// Mitsubishi GX Developer project: 11-702日式面打機_201109261430   PLC: FX1S

PROGRAM MAIN
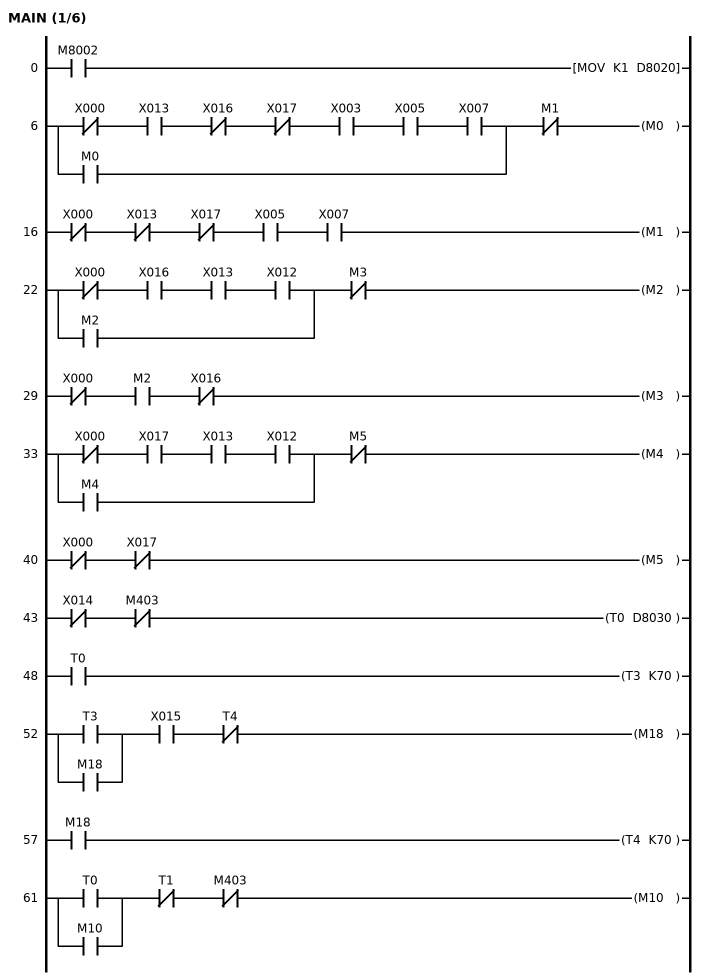
0     LD      M8002
      MOV     K1 D8020
6     LDI     X000
      AND     X013
      ANI     X016
      ANI     X017
      AND     X003
      AND     X005
      AND     X007
      OR      M0
      ANI     M1
      OUT     M0
16    LDI     X000
      ANI     X013
      ANI     X017
      AND     X005
      AND     X007
      OUT     M1
22    LDI     X000
      AND     X016
      AND     X013
      AND     X012
      OR      M2
      ANI     M3
      OUT     M2
29    LDI     X000
      AND     M2
      ANI     X016
      OUT     M3
33    LDI     X000
      AND     X017
      AND     X013
      AND     X012
      OR      M4
      ANI     M5
      OUT     M4
40    LDI     X000
      ANI     X017
      OUT     M5
43    LDI     X014
      ANI     M403
      OUT     T0 D8030
48    LD      T0
      OUT     T3 K70
52    LD      T3
      OR      M18
      AND     X015
      ANI     T4
      OUT     M18
57    LD      M18
      OUT     T4 K70
61    LD      T0
      OR      M10
      ANI     T1
      ANI     M403
      OUT     M10
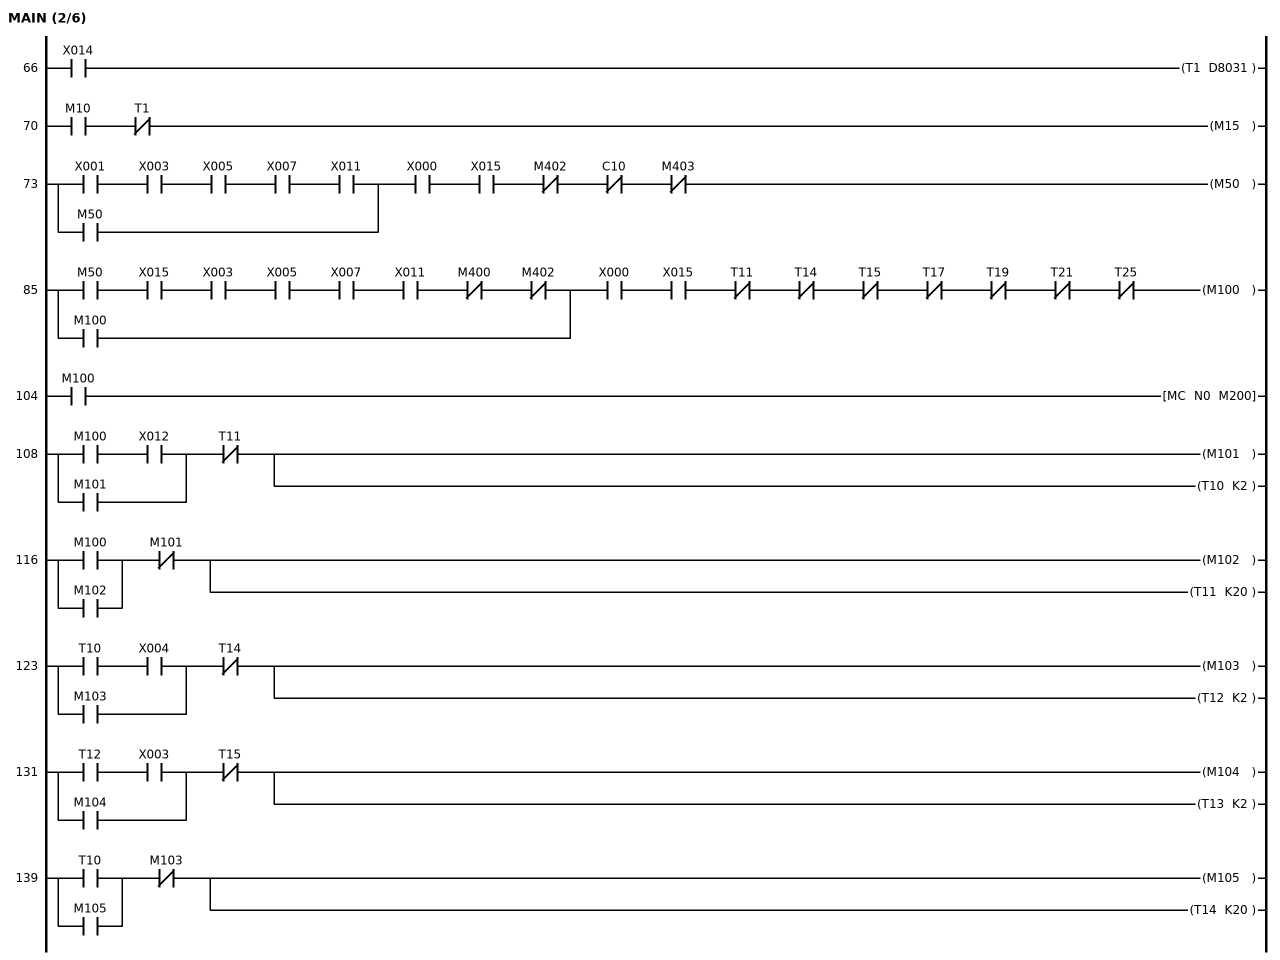
66    LD      X014
      OUT     T1 D8031
70    LD      M10
      ANI     T1
      OUT     M15
73    LD      X001
      AND     X003
      AND     X005
      AND     X007
      AND     X011
      OR      M50
      AND     X000
      AND     X015
      ANI     M402
      ANI     C10
      ANI     M403
      OUT     M50
85    LD      M50
      AND     X015
      AND     X003
      AND     X005
      AND     X007
      AND     X011
      ANI     M400
      ANI     M402
      OR      M100
      AND     X000
      AND     X015
      ANI     T11
      ANI     T14
      ANI     T15
      ANI     T17
      ANI     T19
      ANI     T21
      ANI     T25
      OUT     M100
104   LD      M100
      MC      N0 M200
108   LD      M100
      AND     X012
      OR      M101
      ANI     T11
      OUT     M101
      OUT     T10 K2
116   LD      M100
      OR      M102
      ANI     M101
      OUT     M102
      OUT     T11 K20
123   LD      T10
      AND     X004
      OR      M103
      ANI     T14
      OUT     M103
      OUT     T12 K2
131   LD      T12
      AND     X003
      OR      M104
      ANI     T15
      OUT     M104
      OUT     T13 K2
139   LD      T10
      OR      M105
      ANI     M103
      OUT     M105
      OUT     T14 K20
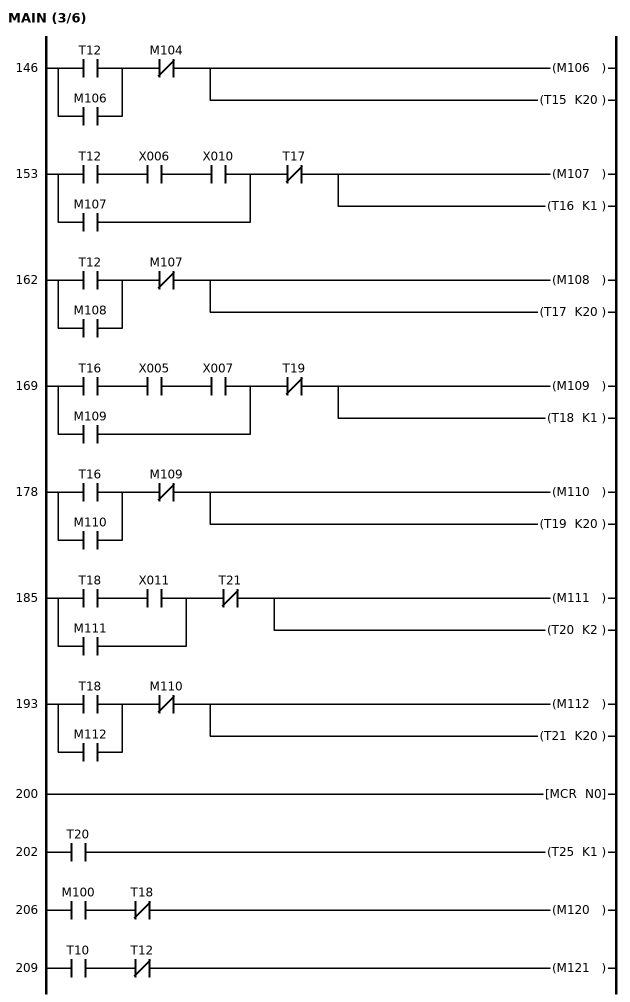
146   LD      T12
      OR      M106
      ANI     M104
      OUT     M106
      OUT     T15 K20
153   LD      T12
      AND     X006
      AND     X010
      OR      M107
      ANI     T17
      OUT     M107
      OUT     T16 K1
162   LD      T12
      OR      M108
      ANI     M107
      OUT     M108
      OUT     T17 K20
169   LD      T16
      AND     X005
      AND     X007
      OR      M109
      ANI     T19
      OUT     M109
      OUT     T18 K1
178   LD      T16
      OR      M110
      ANI     M109
      OUT     M110
      OUT     T19 K20
185   LD      T18
      AND     X011
      OR      M111
      ANI     T21
      OUT     M111
      OUT     T20 K2
193   LD      T18
      OR      M112
      ANI     M110
      OUT     M112
      OUT     T21 K20
200   MCR     N0
202   LD      T20
      OUT     T25 K1
206   LD      M100
      ANI     T18
      OUT     M120
209   LD      T10
      ANI     T12
      OUT     M121
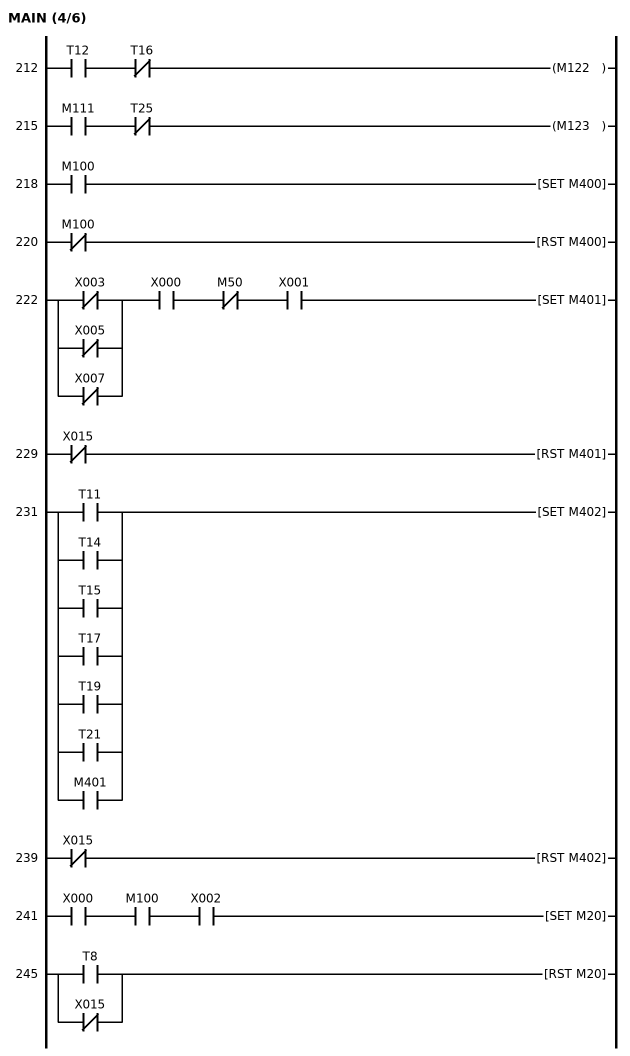
212   LD      T12
      ANI     T16
      OUT     M122
215   LD      M111
      ANI     T25
      OUT     M123
218   LD      M100
      SET     M400
220   LDI     M100
      RST     M400
222   LDI     X003
      ORI     X005
      ORI     X007
      AND     X000
      ANI     M50
      AND     X001
      SET     M401
229   LDI     X015
      RST     M401
231   LD      T11
      OR      T14
      OR      T15
      OR      T17
      OR      T19
      OR      T21
      OR      M401
      SET     M402
239   LDI     X015
      RST     M402
241   LD      X000
      AND     M100
      AND     X002
      SET     M20
245   LD      T8
      ORI     X015
      RST     M20
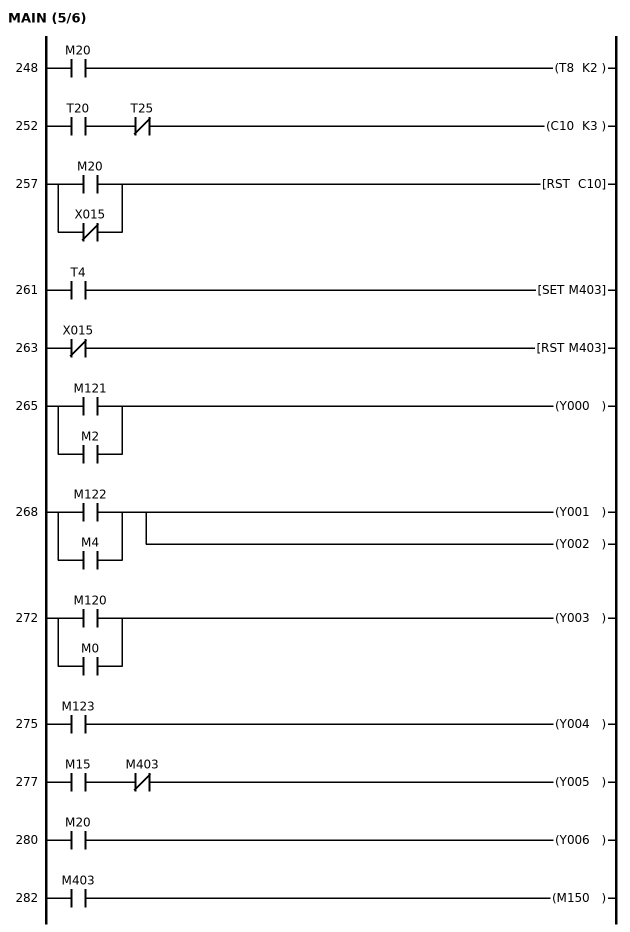
248   LD      M20
      OUT     T8 K2
252   LD      T20
      ANI     T25
      OUT     C10 K3
257   LD      M20
      ORI     X015
      RST     C10
261   LD      T4
      SET     M403
263   LDI     X015
      RST     M403
265   LD      M121
      OR      M2
      OUT     Y000
268   LD      M122
      OR      M4
      OUT     Y001
      OUT     Y002
272   LD      M120
      OR      M0
      OUT     Y003
275   LD      M123
      OUT     Y004
277   LD      M15
      ANI     M403
      OUT     Y005
280   LD      M20
      OUT     Y006
282   LD      M403
      OUT     M150
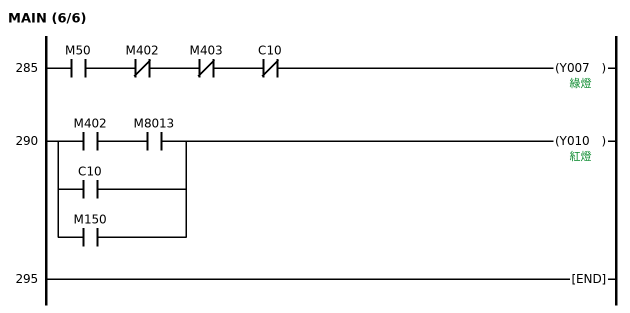
285   LD      M50
      ANI     M402
      ANI     M403
      ANI     C10
      OUT     Y007  ; 綠燈
290   LD      M402
      AND     M8013
      OR      C10
      OR      M150
      OUT     Y010  ; 紅燈
295   END
END_PROGRAM
